{attribute 'GeneratedUsingTerminal: CX2040 EtherCAT slave-1b82-0016'}
{attribute addProperty BoxType "CX2040 EtherCAT slave-1b82-0016"}
{attribute addProperty Description "CX2040 EtherCAT slave"}
{attribute addProperty Physics "YY"}
{attribute addProperty Id "IO_InputsEMPTY_STRUCTURE0Device_Status_MappingAT %I*Device_Status_Mapping_61F790772IO_OutputsEMPTY_STRUCTURE0WcStateAT %I*WcState_9091E0EB2InfoDataAT %I*InfoData_90184F0C16"}
{attribute addProperty CRC "4277641850"}
{attribute addProperty Size "20"}
TYPE CX2040_EtherCAT_slave_FEF7A27A EXTENDS EtcSlaveBoxBase_77A0E4A7 :
STRUCT
	{attribute addProperty Name "IO_Inputs"}
	IO_Inputs : EMPTY_STRUCTURE;
	{attribute addProperty Name "Device_Status_Mapping"}
	Device_Status_Mapping : Device_Status_Mapping_61F79077;
	{attribute addProperty Name "IO_Outputs"}
	IO_Outputs : EMPTY_STRUCTURE;
	{attribute addProperty Name "WcState"}
	WcState : WcState_9091E0EB;
	{attribute addProperty Name "InfoData"}
	InfoData : InfoData_90184F0C;
END_STRUCT
END_TYPE

(* stored: Version 1.2.0.0, ProductVersion 3.1.4024.9
   DUT CX2040_EtherCAT_slave_FEF7A27A: Id {433c350b-86ac-4218-aa30-fc3c1531bc4b} *)
